(* This function block holds results of the complete test run, i.e. results for all test suites *)
FUNCTION_BLOCK FB_TestResults IMPLEMENTS I_TestResults
VAR
    (* Test results *)
    TestSuiteResults : ST_TestSuiteResults;

    (* Misc variables *)
    StoringTestSuiteResultNumber : UINT(1..GVL_Param_TcUnit.MaxNumberOfTestSuites);
    StoringTestSuiteTrigger : Tc2_Standard.R_TRIG;
    StoredTestSuiteResults : BOOL;
    StoredGeneralTestResults : BOOL;
    NumberOfTestsToAnalyse : UINT(1..GVL_Param_TcUnit.MaxNumberOfTestSuites);
END_VAR
VAR_TEMP
    TestSuiteName : Tc2_System.T_MaxString;
    TestName : Tc2_System.T_MaxString;

    TestsInTestSuiteCounter : UINT(1..GVL_Param_TcUnit.MaxNumberOfTestsForEachTestSuite);

    TestToBeStored : FB_Test;
    GeneralTestResultsTestSuitesCounter : UINT(1..GVL_Param_TcUnit.MaxNumberOfTestSuites);
END_VAR

(* The body of the function block stores the test results *)
IF StoringTestSuiteResultNumber <= GVL_TcUnit.NumberOfInitializedTestSuites AND NOT StoredTestSuiteResults THEN
    StoringTestSuiteTrigger(CLK := GVL_TcUnit.TestSuiteAddresses[StoringTestSuiteResultNumber]^.AreAllTestsFinished());
    IF StoringTestSuiteTrigger.Q THEN
        (* Remove everything except the program name + "." + test suite name *)
        TestSuiteName := F_RemoveInstancePathAndProjectNameFromTestInstancePath(TestInstancePath := GVL_TcUnit.TestSuiteAddresses[StoringTestSuiteResultNumber]^.GetInstancePath());

        (* Store test suite name and ID *)
        TestSuiteResults.TestSuiteResults[StoringTestSuiteResultNumber].Name := TestSuiteName;
        TestSuiteResults.TestSuiteResults[StoringTestSuiteResultNumber].Identity := StoringTestSuiteResultNumber - 1;

        (* Store number of tests in test suite *)
        TestSuiteResults.TestSuiteResults[StoringTestSuiteResultNumber].NumberOfTests :=
            GVL_TcUnit.TestSuiteAddresses[StoringTestSuiteResultNumber]^.GetNumberOfTests();

        (* Store number of failed tests in test suite *)
        TestSuiteResults.TestSuiteResults[StoringTestSuiteResultNumber].NumberOfFailedTests :=
            GVL_TcUnit.TestSuiteAddresses[StoringTestSuiteResultNumber]^.GetNumberOfFailedTests();

        (* Limit the test analyse to the max array limit of 'Tests[]' in FB_TestSuite *)
        NumberOfTestsToAnalyse := GVL_TcUnit.TestSuiteAddresses[StoringTestSuiteResultNumber]^.GetNumberOfTestsToAnalyse();

        (* Iterate and print all tests in test suite *)
        FOR TestsInTestSuiteCounter := 1 TO NumberOfTestsToAnalyse BY 1 DO
            TestToBeStored := GVL_TcUnit.TestSuiteAddresses[StoringTestSuiteResultNumber]^.GetTestByPosition(TestsInTestSuiteCounter);
            (* Store test name *)
            TestSuiteResults.TestSuiteResults[StoringTestSuiteResultNumber].TestCaseResults[TestsInTestSuiteCounter].TestName := TestToBeStored.GetName();

            (* Store test class name *)
            TestSuiteResults.TestSuiteResults[StoringTestSuiteResultNumber].TestCaseResults[TestsInTestSuiteCounter].TestClassName :=
                F_RemoveInstancePathAndProjectNameFromTestInstancePath(GVL_TcUnit.TestSuiteAddresses[StoringTestSuiteResultNumber]^.GetInstancePath());

            (* Store whether the test has failed *)
            TestSuiteResults.TestSuiteResults[StoringTestSuiteResultNumber].TestCaseResults[TestsInTestSuiteCounter].TestIsFailed :=
                TestToBeStored.IsFailed();

            (* Store whether the test was skipped *)
            TestSuiteResults.TestSuiteResults[StoringTestSuiteResultNumber].TestCaseResults[TestsInTestSuiteCounter].TestIsSkipped :=
                TestToBeStored.IsSkipped();

            (* Store the (first failed) assertion message *)
            TestSuiteResults.TestSuiteResults[StoringTestSuiteResultNumber].TestCaseResults[TestsInTestSuiteCounter].FailureMessage :=
                TestToBeStored.GetAssertionMessage();

            (* Store the (first failed) assertion type *)
            TestSuiteResults.TestSuiteResults[StoringTestSuiteResultNumber].TestCaseResults[TestsInTestSuiteCounter].FailureType :=
                TestToBeStored.GetAssertionType();

            (* Store number of assertions made *)
            TestSuiteResults.TestSuiteResults[StoringTestSuiteResultNumber].TestCaseResults[TestsInTestSuiteCounter].NumberOfAsserts :=
                TestToBeStored.GetNumberOfAssertions();
        END_FOR

        IF StoringTestSuiteResultNumber = GVL_TcUnit.NumberOfInitializedTestSuites THEN
            StoredTestSuiteResults := TRUE;
        ELSE
            StoringTestSuiteResultNumber := StoringTestSuiteResultNumber + 1;
        END_IF
        StoringTestSuiteTrigger(CLK := FALSE); // Reset trigger
    END_IF
END_IF

(* If all test suites have finished running, store the general test results *)
(* Take care of the special case where no tests have not yet been defined *)
IF GVL_TcUnit.NumberOfInitializedTestSuites = 0 AND (NOT StoredGeneralTestResults) THEN
    StoredGeneralTestResults := TRUE;
    StoredTestSuiteResults := TRUE;
ELSIF StoringTestSuiteResultNumber = GVL_TcUnit.NumberOfInitializedTestSuites AND_THEN
    GVL_TcUnit.TestSuiteAddresses[StoringTestSuiteResultNumber]^.AreAllTestsFinished() AND StoredTestSuiteResults AND (NOT StoredGeneralTestResults) THEN
    TestSuiteResults.NumberOfTestSuites := GVL_TcUnit.NumberOfInitializedTestSuites;
    FOR GeneralTestResultsTestSuitesCounter := 1 TO GVL_TcUnit.NumberOfInitializedTestSuites BY 1 DO
        TestSuiteResults.NumberOfTestCases := TestSuiteResults.NumberOfTestCases + TestSuiteResults.TestSuiteResults[GeneralTestResultsTestSuitesCounter].NumberOfTests;
        TestSuiteResults.NumberOfSuccessfulTestCases := TestSuiteResults.NumberOfSuccessfulTestCases +
                                                        (TestSuiteResults.TestSuiteResults[GeneralTestResultsTestSuitesCounter].NumberOfTests -
                                                         TestSuiteResults.TestSuiteResults[GeneralTestResultsTestSuitesCounter].NumberOfFailedTests);
        TestSuiteResults.NumberOfFailedTestCases := TestSuiteResults.NumberOfFailedTestCases + TestSuiteResults.TestSuiteResults[GeneralTestResultsTestSuitesCounter].NumberOfFailedTests;
    END_FOR
    StoredGeneralTestResults := TRUE;
END_IF

(* Returns whether the storing of the test results is finished *)
METHOD PUBLIC GetAreTestResultsAvailable : BOOL
GetAreTestResultsAvailable := (StoredTestSuiteResults AND StoredGeneralTestResults);
END_METHOD

METHOD PUBLIC GetTestSuiteResults : REFERENCE TO ST_TestSuiteResults;
GetTestSuiteResults REF=TestSuiteResults;
END_METHOD

METHOD ResetTestResult
TestSuiteResults.NumberOfTestSuites				:= 0;
TestSuiteResults.NumberOfTestCases				:= 0;
TestSuiteResults.NumberOfSuccessfulTestCases	:= 0;
TestSuiteResults.NumberOfFailedTestCases		:= 0;

StoringTestSuiteResultNumber	:= 1;
StoredTestSuiteResults			:= FALSE;
StoredGeneralTestResults		:= FALSE;
END_METHOD

END_FUNCTION_BLOCK

(* stored: Version 1.1.0.1, ProductVersion 3.1.4024.11
   POU FB_TestResults: Id {dcfade2b-3801-4064-9466-67a7a848e8d0}, SpecialFunc None
   Method GetAreTestResultsAvailable: Id {1405a17f-835e-481b-8bc4-6f447bc860a2}
   Method GetTestSuiteResults: Id {3d7cfdb1-16a3-456d-be0a-82cecf4820a8}
   Method ResetTestResult: Id {785b1a16-cc1c-4870-a3cd-6e28d350b720} *)
